(* PLC project run, Dassault Systèmes ControlBuild 2024x *)
(* stored: creationDateTime 2023-10-03T11:13:44-01:00 *)

FUNCTION_BLOCK drill.run
  VAR_INPUT
    rotationFault : DINT := 0;
  END_VAR
  VAR_INPUT
    downState : BOOL := false;
    downDeceleration : BOOL := false;
    topDeceleration : BOOL := false;
    topState : BOOL := false;
    motorFault : DINT := 0;
  END_VAR
  VAR_INPUT
    clampingFault : DINT := 0;
    releasingOK : BOOL := false;
    clampingOK : BOOL := false;
  END_VAR
  VAR_INPUT
    emptyProd : BOOL := false;
    unitProd : BOOL := false;
    batchProd : BOOL := false;
  END_VAR
  VAR_INPUT
    acknowledgePB : BOOL := false;
    piece : BOOL := false;
  END_VAR
  VAR_OUTPUT
    rotation : BOOL := false;
    cycleEnd : BOOL := false;
    movementFault : DINT := 0;
    loadingRequest : BOOL := false;
    unloadingRequest : BOOL := false;
    faultyState : BOOL := false;
  END_VAR
  VAR_OUTPUT
    slowAscent : BOOL := false;
    fastAscent : BOOL := false;
    slowDescent : BOOL := false;
    fastDescent : BOOL := false;
  END_VAR
  VAR_OUTPUT
    releasing : BOOL := false;
    clamping : BOOL := false;
  END_VAR
  VAR
    initialCond : BOOL := false;
    noFaultCond : BOOL := false;
    cnt : DINT := 0;
  END_VAR
  VAR CONSTANT
    fastDescentDuration : DINT := 100;
    slowDescentDuration : DINT := 50;
    fastAscentDuration : DINT := 100;
    slowAscentDuration : DINT := 50;
  END_VAR

INITIAL_STEP 10:
  10_INLINE1(N);
  COMPUTE_FUNCTION_BLOCKS(S);
END_STEP
ACTION 10_INLINE1:
  loadingRequest;
  cycleEnd;
END_ACTION
TRANSITION FROM 10 TO 11
  := initialCond;
END_TRANSITION
STEP 11:
  11_INLINE2(N);
END_STEP
ACTION 11_INLINE2:
  clamping;
END_ACTION
TRANSITION FROM 11 TO 12
  := clampingOK;
END_TRANSITION
STEP 12:
  12_INLINE3(N);
END_STEP
ACTION 12_INLINE3:
  fastDescent;
  rotation;
  cnt := cnt + 1;
END_ACTION
TRANSITION FROM 12 TO 13
  := downDeceleration;
END_TRANSITION
STEP 13:
  13_INLINE4(N);
END_STEP
ACTION 13_INLINE4:
  slowDescent;
  rotation;
  cnt := cnt + 1;
END_ACTION
TRANSITION FROM 13 TO 14
  := downState;
END_TRANSITION
STEP 14:
  14_INLINE5(N);
END_STEP
ACTION 14_INLINE5:
  fastAscent;
  rotation;
  cnt := cnt + 1;
END_ACTION
TRANSITION FROM 14 TO 15
  := topDeceleration;
END_TRANSITION
STEP 15:
  15_INLINE6(N);
END_STEP
ACTION 15_INLINE6:
  slowAscent;
  cnt := cnt + 1;
END_ACTION
TRANSITION FROM 15 TO 16
  := topState;
END_TRANSITION
STEP 16:
  16_INLINE7(N);
END_STEP
ACTION 16_INLINE7:
  releasing;
END_ACTION
TRANSITION FROM 16 TO 17
  := releasingOK;
END_TRANSITION
STEP 17:
  17_INLINE8(N);
END_STEP
ACTION 17_INLINE8:
  cycleEnd;
  unloadingRequest;
END_ACTION
TRANSITION FROM 17 TO 10
  := NOT piece;
END_TRANSITION
ACTION COMPUTE_FUNCTION_BLOCKS:  (* blocks drawn on the SFC sheet *)
  G1:
END_ACTION

ACTION PreSFC:
IF(RE acknowledgePB) THEN
	movementFault := 0;
END_IF;
IF((X12 AND (cnt >= fastDescentDuration)  AND NOT downDeceleration )) THEN
	movementFault := 1;
END_IF;
IF((X13 AND (cnt >= slowDescentDuration)  AND NOT downState )) THEN
	movementFault := 2;
END_IF;
IF((X14 AND (cnt >= fastAscentDuration)  AND NOT topDeceleration )) THEN
	movementFault := 3;
END_IF;
IF((X15 AND (cnt >= slowAscentDuration)  AND NOT topState )) THEN
	movementFault := 4;
END_IF;
IF((X12 AND downState  AND NOT downDeceleration )) THEN
	movementFault := 5;
END_IF;
IF((X14 AND topState  AND NOT topDeceleration )) THEN
	movementFault := 6;
END_IF;
IF(((X13 OR X14) AND topState )) THEN
	movementFault := 7;
END_IF;
IF(((X11 OR X13 OR X16 OR X17) AND topDeceleration )) THEN
	movementFault := 8;
END_IF;
IF(((X11 OR X15 OR X16 OR X17) AND downDeceleration )) THEN
	movementFault := 9;
END_IF;
IF(((X11 OR X15 OR X16 OR X17) AND downState )) THEN
	movementFault := 10;
END_IF;
noFaultCond := (clampingFault = 0) AND (motorFault = 0)  AND (rotationFault = 0)  AND (movementFault = 0) ;
initialCond := noFaultCond AND ((piece AND (RE unitProd OR batchProd) ) OR emptyProd) ;
END_ACTION

ACTION PostSFC:
IF((X10 OR RE X12 OR RE X13 OR RE X14 OR RE X15)) THEN
	cnt := 0;
END_IF;
faultyState := NOT noFaultCond;
END_ACTION
END_FUNCTION_BLOCK
